TYPE DUT_SENSOR_DATAS_h3 :
UNION
	data_lreal:REAL;
	data_byte:ARRAY[0..3] OF BYTE;
END_UNION
END_TYPE

(* stored: Version 1.1.0.1, ProductVersion 3.1.4024.6
   DUT DUT_SENSOR_DATAS_h3: Id {4a35e2ee-825e-40b7-9764-3e5535b375b0} *)
